(* CODESYS project I2C_EncoderEmulator.library
   Author: Open Source
   Version: 1.0.0.0
   Description: An I/O driver template, meant to easily map an existing FB to the CODESYS I/O driver interface
   Title: I2C_EncoderEmulator
   DefaultNamespace: I2C_EncoderEmulator
   Placeholder: SPI MCP3008
   Company: Open Source

Project tree, tasks and I/O mapping:
  libraries: Standard, * (System); IoStandard, * (System); IoDrvBase, * (System); IoDriver Parameter Interfaces, * (System); IoDriver Interfaces, * (System); CmpErrors2 Interfaces, * (System); SysTypes2 Interfaces, * (System); Raspberry Pi Peripherals, 3.5.11.0 (3S - Smart Software Solutions GmbH)
  00000000-0000-0000-0000-000000000000|D:\CoDeSys\LibrariesV3\trunk\Intern\CAA\CAA Template\3.2.0.3 draft\Prefix.pdf
  00000000-0000-0000-0000-000000000000|D:\CoDeSys\LibrariesV3\trunk\Intern\CAA\CAA Template\3.4.0.0 draft\Placeholder.xml
  00000000-0000-0000-0000-000000000000|D:\CoDeSys\LibrariesV3\trunk\Intern\CAA\CAA Template\3.5.2.0 draft\Placeholder.xml
  global variables GVL
  Generic/
    function block IoDrvI2CEncoderEmulator [ST]: FB_Init, Initialize, QueryInterface, FB_Exit, FB_Reinit, IoDrvReadInputs, IoDrvStartBusCycle, IoDrvUpdateConfiguration, IoDrvWriteOutputs, IoDrvGetModuleDiagnosis, IoDrvUpdateMapping, IoDrvWatchdogTrigger, IoDrvIdentify, IoDrvScanModules, IoDrvReadParameter, IoDrvWriteParameter, IoDrvGetConnector
  function block I2CEncoderEmulator [ST]: AfterReadInputs, BeforeWriteOutputs, Initialize
*)

// GVL
VAR_GLOBAL CONSTANT
	cClassID: DWORD := 16#0003FFFF;
	cDriverName : STRING(31) := 'IoDrvFB';
	cDeviceName : STRING(31) := 'IoDrvFB';
	cVendorName : STRING(31) := 'Open Source';
	cModuleType : WORD := 8007;
END_VAR

// Generic/IoDrvI2CEncoderEmulator
FUNCTION_BLOCK IoDrvI2CEncoderEmulator EXTENDS IoDrvBase IMPLEMENTS ICmpIoDrvParameter
VAR_INPUT
END_VAR
VAR_OUTPUT
END_VAR
VAR CONSTANT
	CLASSID_CCmpIoDrvTemplate : DWORD := 16#0000FF03; //TODO
END_VAR
VAR
	_IIoDrv : ICmpIoDrv;
	_IIoDrvParameter : ICmpIoDrvParameter;
	_instance: I2CEncoderEmulator;
	_xBackGroundDiagStarted : BOOL;

END_VAR

{attribute 'conditionalshow'}
METHOD FB_Init : BOOL
VAR_INPUT
	bInitRetains : BOOL;
	bInCopyCode : BOOL;
END_VAR
VAR
	Result : UDINT;
END_VAR
FB_Init_Count := FB_Init_Count + 1;

m_Info.szDriverName := cDriverName;
m_Info.szVendorName := cVendorName;
m_info.szDeviceName := cDeviceName;
m_Info.wModuleType := cModuleType;

_IIoDrv := THIS^;
_IIoDrvParameter := THIS^;

m_IBaseItf := THIS^;
m_hInterface := IoMgrRegisterInstance2(dwClassId:=CLASSID_CCmpIoDrvTemplate(*cClassID*), pItf:=m_IBaseItf, pResult:=ADR(Result));
FB_Init := TRUE;
END_METHOD

{attribute 'conditionalshow'}
METHOD Initialize : UDINT
VAR_INPUT
	wModuleType : UINT;
	dwInstance : UDINT;
	pConnector : POINTER TO IoConfigConnector; 
END_VAR
VAR
END_VAR
Initialize_Count := Initialize_Count + 1;

m_wModuleType := wModuleType;
m_dwInstance := dwInstance;
m_Info.wModuleType := wModuleType;

_Instance.Initialize(wModuleType, dwInstance, pConnector);

Initialize := CmpErrors.Errors.ERR_OK;
END_METHOD

{attribute 'conditionalshow'}
METHOD QueryInterface : POINTER TO POINTER TO BYTE
VAR_INPUT
	iid : DWORD; (* InterfaceID *)
	pResult : POINTER TO UDINT;	
END_VAR
VAR
END_VAR
IF iid = ITFID_ICmpIoDrv THEN
	QueryInterface := ADR(_IIoDrv);
	AddRef();
	IF (pResult <> 0) THEN
		pResult^ := Errors.ERR_OK;
	END_IF
	RETURN;	
ELSIF iid = ITFID_ICmpIoDrvParameter THEN
	QueryInterface := ADR(_IIoDrvParameter);
	AddRef();
	IF (pResult <> 0) THEN
		pResult^ := Errors.ERR_OK;
	END_IF	
	RETURN;	
ELSE
	QueryInterface := SUPER^.QueryInterface(iid, pResult);
END_IF
END_METHOD

{attribute 'conditionalshow'}
METHOD FB_Exit : Bool
VAR_INPUT
	bInCopyCode : BOOL;
END_VAR
FB_Exit_Count := FB_Exit_Count + 1;
FB_Exit := TRUE;
END_METHOD

{attribute 'conditionalshow'}
METHOD FB_Reinit : BOOL
VAR_INPUT
END_VAR
VAR
END_VAR
FB_Reinit_Count := FB_Reinit_Count + 1;
FB_Reinit := TRUE;
END_METHOD

{attribute 'conditionalshow'}
METHOD IoDrvReadInputs : UDINT
VAR_INPUT
	pConnectorMapList : POINTER TO IoConfigConnectorMap;
	nCount : DINT;
END_VAR
VAR
	i, j : DINT;
END_VAR
IF pConnectorMapList = 0 OR nCount = 0 THEN
	IoDrvReadInputs := Errors.ERR_PARAMETER;
	RETURN;
END_IF

FOR i:=0 TO nCount - 1 DO
	IF (pConnectorMapList[i].dwNumOfChannels = 0) THEN
		CONTINUE;
	END_IF
	FOR j:= 0 TO UDINT_TO_UINT(pConnectorMapList[i].dwNumOfChannels) - 1 DO	
		IoMgrCopyInputLE(ADR(pConnectorMapList[i].pChannelMapList[j]), pConnectorMapList[i].pChannelMapList[j].pParameter^.dwDriverSpecific);
	END_FOR
END_FOR

IoDrvReadInputs := Errors.ERR_OK;
END_METHOD

{attribute 'conditionalshow'}
METHOD IoDrvStartBusCycle : UDINT
VAR_INPUT
	pConnector : POINTER TO IoConfigConnector;
END_VAR
VAR
END_VAR
_instance();

IoDrvStartBusCycle := Errors.ERR_OK;
END_METHOD

{attribute 'conditionalshow'}
METHOD IoDrvUpdateConfiguration : UDINT
VAR_INPUT
	pConnectorList : POINTER TO IoConfigConnector;
	nCount : DINT;
END_VAR
VAR
	pParameter : POINTER TO IoConfigParameter;	
	Result : RTS_IEC_RESULT;
	pudtConfig : POINTER TO IoDrvConfig;
END_VAR
IoDrvUpdateConfiguration_Count := IoDrvUpdateConfiguration_Count + 1;
IoDrvUpdateConfiguration := Errors.ERR_OK;

IF (pConnectorList = 0) THEN
	RETURN;
END_IF

m_pConnector := IoMgrConfigGetConnector(pConnectorList, ADR(nCount), m_wModuleType, m_dwInstance);

IF m_pConnector = 0 THEN
	IoDrvUpdateConfiguration := ERRORS.ERR_PARAMETER;
	RETURN;
END_IF

//check if device is enabled in the device tree
IF (m_pConnector^.dwFlags AND ConnectorFlags.CF_ENABLE) = 0 THEN
	IoDrvUpdateConfiguration := Errors.ERR_OK;
	RETURN;
END_IF

IF m_pConnector^.hIoDrv = 0 THEN
	m_pConnector^.hIoDrv := m_hInterface;
	m_pConnector^.pFather^.hIoDrv := m_hInterface;
	
	{IF defined (pou:IoMgrConfigSetDiagnosis)}
	IoMgrConfigSetDiagnosis(m_pConnector,
							ConnectorFlags.CF_DRIVER_AVAILABLE OR
							ConnectorFlags.CF_CONNECTOR_FOUND OR
							ConnectorFlags.CF_CONNECTOR_CONFIGURED OR
							ConnectorFlags.CF_CONNECTOR_ACTIVE);
	{END_IF}
	
	{IF defined (pou:IoMgrConfigSetDiagnosis)}
	IoMgrConfigSetDiagnosis(m_pConnector^.pFather,
							ConnectorFlags.CF_DRIVER_AVAILABLE OR
							ConnectorFlags.CF_CONNECTOR_FOUND OR
							ConnectorFlags.CF_CONNECTOR_CONFIGURED OR
							ConnectorFlags.CF_CONNECTOR_ACTIVE);
	{END_IF}

	{IF defined (pou:IoMgrSetDriverProperties)}			
		IoMgrSetDriverProperties(m_hInterface, DRVPROP_CONSISTENCY OR DRVPROP_BACKGROUND_GETDIAG);
	{END_IF}										

	// Map config-, input- and output parameters
	(*pParameter := IoMgrConfigGetParameter(m_pConnector, 1000);
	IF (pParameter <> 0) THEN
		pParameter^.dwDriverSpecific := ADR(_instance.udtInput);
	END_IF
	*)
	pParameter := IoMgrConfigGetParameter(m_pConnector, 2000);
	IF (pParameter <> 0) THEN
		pParameter^.dwDriverSpecific := ADR(_instance.cmd);
	END_IF
	pParameter := IoMgrConfigGetParameter(m_pConnector, 2001);
	IF (pParameter <> 0) THEN
		pParameter^.dwDriverSpecific := ADR(_instance.rpm);
	END_IF
	pParameter := IoMgrConfigGetParameter(m_pConnector, 2002);
	IF (pParameter <> 0) THEN
		pParameter^.dwDriverSpecific := ADR(_instance.resolucao);
	END_IF

	pParameter := IoMgrConfigGetParameter(m_pConnector, 3000);
	IF (pParameter <> 0) THEN
		pudtConfig := IoStandard.ConfigGetParameterValuePointer(pParameter, ADR(Result));
		_instance.usiAddress := pudtConfig^;
	END_IF
END_IF
END_METHOD

{attribute 'conditionalshow'}
METHOD IoDrvWriteOutputs : UDINT
VAR_INPUT
	pConnectorMapList : POINTER TO IoConfigConnectorMap;
	nCount : DINT;
END_VAR
VAR
	i, j : DINT;
	pbyIecAddress : POINTER TO BYTE;
	wSrcIndex : WORD;	
	wDestIndex : WORD;	
	ptrBy: POINTER TO BYTE;
	ptrW: POINTER TO BYTE;

END_VAR
IF pConnectorMapList = 0 OR nCount = 0 THEN
	IoDrvWriteOutputs := Errors.ERR_PARAMETER;
	RETURN;
END_IF

FOR i:=0 TO nCount - 1 DO
	IF (pConnectorMapList[i].dwNumOfChannels = 0) THEN
		CONTINUE;
	END_IF
	FOR j:= 0 TO UDINT_TO_UINT(pConnectorMapList[i].dwNumOfChannels) - 1 DO	
		IoMgrCopyOutputLE(ADR(pConnectorMapList[i].pChannelMapList[j]), pConnectorMapList[i].pChannelMapList[j].pParameter^.dwDriverSpecific);
		(*wSrcIndex := pConnectorMapList[i].pChannelMapList[j].wIecAddressBitOffset / 8; 
		pbyIecAddress := pConnectorMapList[i].pChannelMapList[j].pbyIecAddress;
		IF pConnectorMapList[i].pChannelMapList[j].pParameter^.dwParameterId = 2000 THEN		
			IF pConnectorMapList[i].pChannelMapList[j].wSize = 8 THEN
				ptrBy:= pbyIecAddress;
				_instance.cmd := ptrBy^;
			END_IF
		ELSIF pConnectorMapList[i].pChannelMapList[j].pParameter^.dwParameterId = 2001 THEN		
			IF pConnectorMapList[i].pChannelMapList[j].wSize = 16 THEN
				ptrW:= pbyIecAddress;
				_instance.rpm := ptrW^;
			END_IF
		ELSIF pConnectorMapList[i].pChannelMapList[j].pParameter^.dwParameterId = 2002 THEN		
			IF pConnectorMapList[i].pChannelMapList[j].wSize = 16 THEN
				ptrW:= pbyIecAddress;
				_instance.resolucao := ptrW^;
			END_IF
		END_IF;*)
	END_FOR
END_FOR
END_METHOD

METHOD IoDrvGetModuleDiagnosis : UDINT
VAR_INPUT
	pConnector : POINTER TO IoConfigConnector;
END_VAR
VAR
END_VAR
IF pConnector = 0 THEN
	//we are called from the background task
	_xBackGroundDiagStarted := TRUE;
END_IF

//Todo: update connectorflags if something changed

IoDrvGetModuleDiagnosis_Count := IoDrvGetModuleDiagnosis_Count + 1;
IoDrvGetModuleDiagnosis := Errors.ERR_NOTIMPLEMENTED;
END_METHOD

METHOD IoDrvUpdateMapping : UDINT
VAR_INPUT
	pTaskMapList : POINTER TO IoConfigTaskMap;
	nCount : DINT;	
END_VAR
VAR
END_VAR
IoDrvUpdateMapping_Count := IoDrvUpdateMapping_Count + 1;

IF (pTaskMapList = 0) THEN
	IoDrvUpdateMapping := Errors.ERR_PARAMETER;
	RETURN;
END_IF

IoDrvUpdateMapping := Errors.ERR_OK;
END_METHOD

METHOD IoDrvWatchdogTrigger : UDINT
VAR_INPUT
	pConnector : POINTER TO IoConfigConnector;	
END_VAR
VAR
END_VAR
IoDrvWatchdogTrigger_Count := IoDrvWatchdogTrigger_Count + 1;
IoDrvWatchdogTrigger := Errors.ERR_OK;
END_METHOD

METHOD IoDrvIdentify : UDINT
VAR_INPUT
	pConnector : POINTER TO IoConfigConnector;	
END_VAR
VAR
END_VAR
IoDrvIdentify_Count := IoDrvIdentify_Count + 1;
IoDrvIdentify := Errors.ERR_NOTIMPLEMENTED;
END_METHOD

METHOD IoDrvScanModules : UDINT
VAR_INPUT
	pConnector : POINTER TO IoConfigConnector;
	ppConnectorList : POINTER TO POINTER TO IoConfigConnector;
	pnCount : POINTER TO DINT;	
END_VAR
VAR
END_VAR
IoDrvScanModules_Count := IoDrvScanModules_Count + 1;
IoDrvScanModules := Errors.ERR_NOTIMPLEMENTED;
END_METHOD

{attribute 'conditionalshow'}
METHOD IoDrvReadParameter : UDINT
VAR_INPUT
	pConnector : POINTER TO IoConfigConnector;
	pParameter : POINTER TO IoConfigParameter;
	pData : POINTER TO BYTE;
	dwBitSize : DWORD;
	dwBitOffset : DWORD;
END_VAR
VAR
END_VAR
IF 	pConnector = 0 OR pParameter = 0 OR pData = 0 THEN
	IoDrvReadParameter := Errors.ERR_PARAMETER;
	RETURN;	
END_IF

// All standard parameters of our device are handled by the IO-manager!
IoDrvReadParameter := Errors.ERR_FAILED;
END_METHOD

{attribute 'conditionalshow'}
METHOD IoDrvWriteParameter : UDINT
VAR_INPUT
	pConnector : POINTER TO IoConfigConnector;
	pParameter : POINTER TO IoConfigParameter;
	pData : POINTER TO BYTE;
	dwBitSize : DWORD;
	dwBitOffset : DWORD;
END_VAR
VAR
	pParam : POINTER TO IoConfigParameter;
	pstDiagString : POINTER TO STRING;
END_VAR
IF pConnector = 0 OR pParameter = 0 OR pData = 0 THEN
	IoDrvWriteParameter := Errors.ERR_PARAMETER;
	RETURN;	
END_IF

IoDrvWriteParameter := Errors.ERR_FAILED;
END_METHOD

METHOD IoDrvGetConnector : POINTER TO IoConfigConnector
VAR_INPUT
	pResult : POINTER TO RTS_IEC_RESULT;
END_VAR
VAR
END_VAR
IF m_pConnector = 0 THEN
	IF pResult <> 0 THEN
		pResult^ := Errors.ERR_FAILED;
	END_IF
	IoDrvGetConnector := 0;	
	RETURN;
END_IF
IF pResult <> 0 THEN
	pResult^ := Errors.ERR_OK;
END_IF
IoDrvGetConnector := m_pConnector;
END_METHOD

END_FUNCTION_BLOCK

// I2CEncoderEmulator
FUNCTION_BLOCK I2CEncoderEmulator EXTENDS i2c
VAR_INPUT
	cmd : BYTE;
	rpm : UINT;
	resolucao	: UINT;
END_VAR
VAR
	timer: TON := (IN:=TRUE);
	_temp	: WORD;
END_VAR

SUPER^();

CASE _iState OF
0:
	(*IF usiAddress = 0 THEN
		usiAddress := udtConfig.usiAddress;
	END_IF*)
	IF SUPER^.init() THEN
		_iState := 5;
	END_IF	

5:	
	Timer.pt := T#70MS;
	_iState := 10;	
END_CASE

METHOD AfterReadInputs : INT
VAR
	Buffer : ARRAY[0..4] OF BYTE;
	len: dINT;
END_VAR
SUPER^.AfterReadInputs();

IF _iState = 10 THEN
	timer(IN:=TRUE);
	IF timer.Q THEN	
		Buffer[0]:= cmd;
		Buffer[1]:= WORD_TO_BYTE(SHR(INT_TO_WORD(rpm),8));
		Buffer[2]:= INT_TO_BYTE(rpm);
		Buffer[3]:= WORD_TO_BYTE(SHR(INT_TO_WORD(resolucao),8));
		Buffer[4]:= INT_TO_BYTE(resolucao);
		Write(ADR(Buffer), SIZEOF(Buffer));
		timer(IN:=FALSE);
	END_IF		
END_IF
END_METHOD

METHOD BeforeWriteOutputs : INT
VAR
END_VAR
SUPER^.BeforeWriteOutputs();
END_METHOD

METHOD Initialize : UDINT
VAR_INPUT
	wModuleType : UINT;
	dwInstance : UDINT;
	pConnector : POINTER TO IoConfigConnector;
END_VAR
VAR
	pParam: POINTER TO IoConfigParameter;		
	udiResult: UDINT;
END_VAR
SUPER^.Initialize(wModuleType, dwInstance, pConnector);

pParam := ConfigGetParameter(_pConnector, 3000);
IF pParam <> 0 THEN
	usiAddress := IoStandard.ConfigGetParameterValueByte(pParam, ADR(udiResult));
END_IF

(* no longer supported
pParam := ConfigGetParameter(_pConnector, 3);
IF pParam <> 0 THEN
	_usiUsedOutputs := IoStandard.ConfigGetParameterValueByte(pParam, ADR(udiResult));
END_IF
*)
(*
pParam := ConfigGetParameter(_pConnector, 1);
IF pParam <> 0 THEN	//store own pointer in this param
	pParam^.dwDriverSpecific := THIS;
END_IF

*)
END_METHOD

END_FUNCTION_BLOCK
